TYPE ST_VisionProcessConfig :
STRUCT
    tDetectionDelay : TIME;
    fAngleCorrection : LREAL;
END_STRUCT
END_TYPE

(* stored: Version 1.1.0.1, ProductVersion 3.1.4026.20
   DUT ST_VisionProcessConfig: Id {42274acc-75c3-4a04-812c-ebbc4875d172} *)
